FUNCTION_BLOCK ABSTRACT FB_PositionSensorObserverBase EXTENDS ZigaLibs_Core.FB_HasInstanceName

VAR
	_topPositionObserver 	: ZigaLibs_Core.BoolEx;
	_topPositionError		: Tc2_Standard.R_TRIG;
	
	_bottoPositionObserver	: ZigaLibs_Core.BoolEx;
	_bottomPositionError	: Tc2_Standard.R_TRIG;
	
	_logger					: ZigaLibs_Core.I_LoggerEx;
	_sb						: ZigaLibs_Core.FB_StringBuilder;
END_VAR

VAR
	{attribute 'hide'}
	_topPositionSensor		: BOOL;
	{attribute 'hide'}
	_bottomPositionSensor	: BOOL;
END_VAR

VAR CONSTANT
	MAXIMUM_DURATION_AT_BOTTOM_POSITION : TIME := T#10S;
	MAXIMUM_DURATION_AT_TOP_POSITION 	: TIME := T#10S;
END_VAR

_topPositionObserver(variable := TopPositionSensor);
_bottoPositionObserver(variable := BottomPositionSensor);
_topPositionError(CLK := _topPositionObserver.HasBeenTrueForAtLeast(MAXIMUM_DURATION_AT_TOP_POSITION));
_bottomPositionError(CLK := _bottoPositionObserver.HasBeenTrueForAtLeast(MAXIMUM_DURATION_AT_BOTTOM_POSITION));

PROPERTY BottomPositionSensor : REFERENCE TO BOOL
GET
BottomPositionSensor REF= _bottomPositionSensor;
END_GET
SET
_bottomPositionSensor := BottomPositionSensor;
END_SET
END_PROPERTY

PROPERTY TopPositionSensor : REFERENCE TO BOOL
GET
TopPositionSensor REF= _topPositionSensor;
END_GET
SET
_topPositionSensor := TopPositionSensor;
END_SET
END_PROPERTY

END_FUNCTION_BLOCK

(* stored: Version 1.1.0.1, ProductVersion 3.1.4024.14
   POU FB_PositionSensorObserverBase: Id {2ab8856f-e4f4-0529-1efd-e2a591634266}, SpecialFunc None
   Property BottomPositionSensor: Id {45ba5b9d-ffef-09d6-0dc3-4f2f5b861e26}
   Get Get: Id {5eb07ddd-020d-0fcb-0f9f-2301d15eb2b5}
   Set Set: Id {eaff412f-b5cd-048f-2e6b-cf6ad53d26a9}
   Property TopPositionSensor: Id {686a2265-43ce-0c22-2f7a-998313a90f37}
   Get Get: Id {b0cdeef8-4973-02c4-2d92-64be248ebdcf}
   Set Set: Id {a15de8f0-c7d2-0cca-33da-dc4ee9cff5b1} *)
